// TwinCAT 3 PLC project Untitled1
// ProgramVersion: 3.1.4023.0
// libraries:
//   Tc2_MC2, * (Beckhoff Automation GmbH)
//   Tc2_Standard, * (Beckhoff Automation GmbH)
//   Tc2_System, * (Beckhoff Automation GmbH)
//   Tc3_Module, * (Beckhoff Automation GmbH)
// project tree:
//   DUTs/ stCondition.TcDUT
//   / PlcTask.TcTTO
//   POUs/ MAIN.TcPOU
// real-time tasks:
//   TASK PlcTask: cycle T#10ms, priority 20, ADS port 350
// motion (NC):
//   TASK NC-Task 1 SAF: cycle T#2ms, priority 4, ADS port 501
//   TASK NC-Task 1 SVB: cycle T#10ms, priority 8, ADS port 511
//   AXIS Axis 1 (id 1)
//     OtherSettings: AllowMotionCmdToSlave=true
//     encoder EncType=1
//     drive DrvType=5
//       Analog: TorqueSetpointScale=10, ScaleFactorActTorque=0.1
//     controller CtrType=1
//       CtrPara: PriorControlFactor=1
//         Observer: BandWidth=20
// variable links:
//   Untitled1/Untitled1 Instance <-> NC-Task 1 SAF/Axes/Axis 1
//     PlcTask Inputs/MAIN.fbAxis.NcToPlc <-> Outputs/ToPlc
//     PlcTask Outputs/MAIN.fbAxis.PlcToNc <-> Inputs/FromPlc

CONFIGURATION Untitled1
    RESOURCE PLC ON TwinCAT3
        TASK PlcTask(INTERVAL := T#10ms, PRIORITY := 20);
        PROGRAM MAIN WITH PlcTask : MAIN;
    END_RESOURCE
END_CONFIGURATION

// ---- DUTs/stCondition.TcDUT
TYPE stCondition :
STRUCT
	lrVelocity			: LREAL;
	lrAcceleration		: LREAL;
	lrDeceleration		: LREAL;
	lrJerk				: LREAL;
END_STRUCT
END_TYPE

// ---- POUs/MAIN.TcPOU
PROGRAM MAIN
VAR
	fbAxis						: AXIS_REF;
	fbPower						: MC_Power;
	fbMoveAbs_AC				: MC_MoveAbsolute;
	fbMoveAbs_CD				: MC_MoveAbsolute;
	fbMoveAbs_DE				: MC_MoveAbsolute;
	fbMoveAbs_EB				: MC_MoveAbsolute;
	fbMoveAbs_BA				: MC_MoveAbsolute;
	
	stFastCondition				: stCondition;
	stSlowCondition				: stCondition;
	
	iState						: UINT;
	bInitialized				: BOOL;
	bStartMove					: BOOL;
	
	bExeMoveAbs_AC				: BOOL;
	bExeMoveAbs_CD				: BOOL;
	bExeMoveAbs_DE				: BOOL;
	bExeMoveAbs_EB				: BOOL;
	bExeMoveAbs_BA				: BOOL;
	lrTargetPos_B				: LREAL := 500;					
END_VAR

CASE iState OF
	0: //初期化を始めますか
	IF bInitialized THEN
		iState := 10;
	END_IF
	
	10: //条件を設定します
	iState := 20;
	stFastCondition.lrVelocity := 100;
	stFastCondition.lrAcceleration := 1000;
	stFastCondition.lrDeceleration := 1000;
	stFastCondition.lrJerk := 10000;
	
	stSlowCondition.lrVelocity := 50;
	stSlowCondition.lrAcceleration := 500;
	stSlowCondition.lrDeceleration := 500;
	stSlowCondition.lrJerk := 5000;

	20: // サーボオンします
	fbPower(
		Axis:= fbAxis, 
		Enable:= TRUE, 
		Enable_Positive:= TRUE, 
		Enable_Negative:= TRUE, 
		Override:= , 
		BufferMode:= , 
		Options:= );
		
	IF fbPower.Status THEN
		//サーボオンしたら次へ
		iState := 100;
	END_IF
		
	100: //動作を開始しますか
	IF bStartMove THEN
		iState := 110;
	END_IF
	
	110: 
	IF (-0.1 < fbAxis.NcToPlc.ActPos) AND (fbAxis.NcToPlc.ActPos < 0.1) THEN
		//初期地点でAからCに移動
		bExeMoveAbs_AC := TRUE;
		bExeMoveAbs_CD := FALSE;
		bExeMoveAbs_DE := FALSE;
		bExeMoveAbs_EB := FALSE;
		bExeMoveAbs_BA := FALSE;
	ELSIF (100 < fbAxis.NcToPlc.ActPos) AND (fbAxis.NcToPlc.ActPos < 200) THEN
		// C地点についたら条件を変えてD地点に移動
		bExeMoveAbs_AC := FALSE;
		bExeMoveAbs_CD := TRUE;
		bExeMoveAbs_DE := FALSE;
		bExeMoveAbs_EB := FALSE;
		bExeMoveAbs_BA := FALSE;
	ELSIF (200 < fbAxis.NcToPlc.ActPos) AND (fbAxis.NcToPlc.ActPos < 300) THEN
		// D地点についたら条件を変えてE地点に移動
		bExeMoveAbs_AC := FALSE;
		bExeMoveAbs_CD := FALSE;
		bExeMoveAbs_DE := TRUE;
		bExeMoveAbs_EB := FALSE;
		bExeMoveAbs_BA := FALSE;
	ELSIF (300 < fbAxis.NcToPlc.ActPos) AND (fbAxis.NcToPlc.ActPos < 400) THEN
		// E地点についたら条件を変えてB地点に移動
		bExeMoveAbs_AC := FALSE;
		bExeMoveAbs_CD := FALSE;
		bExeMoveAbs_DE := FALSE;
		bExeMoveAbs_EB := TRUE;
		bExeMoveAbs_BA := FALSE;
	END_IF
	
	IF fbMoveAbs_EB.Done THEN
		//Bに到着
		iState := 120;
	END_IF

// A>C 高速条件
	fbMoveAbs_AC(
		Axis:= fbAxis, 
		Execute:= bExeMoveAbs_AC, 
		Position:= lrTargetPos_B, 
		Velocity:= stFastCondition.lrVelocity, 
		Acceleration:= stFastCondition.lrAcceleration, 
		Deceleration:= stFastCondition.lrDeceleration, 
		Jerk:= stFastCondition.lrJerk, 
		BufferMode:= , 
		Options:= );
		
	// C>D 低速条件
	fbMoveAbs_CD(
		Axis:= fbAxis, 
		Execute:= bExeMoveAbs_CD, 
		Position:= lrTargetPos_B, 
		Velocity:= stSlowCondition.lrVelocity, 
		Acceleration:= stSlowCondition.lrAcceleration, 
		Deceleration:= stSlowCondition.lrDeceleration, 
		Jerk:= stSlowCondition.lrJerk, 
		BufferMode:= , 
		Options:= );
		
	// D>E 高速条件
	fbMoveAbs_DE(
		Axis:= fbAxis, 
		Execute:= bExeMoveAbs_DE, 
		Position:= lrTargetPos_B, 
		Velocity:= stFastCondition.lrVelocity, 
		Acceleration:= stFastCondition.lrAcceleration, 
		Deceleration:= stFastCondition.lrDeceleration, 
		Jerk:= stFastCondition.lrJerk, 
		BufferMode:= , 
		Options:= );
		
	// E>B 低速条件
	fbMoveAbs_EB(
		Axis:= fbAxis, 
		Execute:= bExeMoveAbs_EB, 
		Position:= lrTargetPos_B, 
		Velocity:= stSlowCondition.lrVelocity, 
		Acceleration:= stSlowCondition.lrAcceleration, 
		Deceleration:= stSlowCondition.lrDeceleration, 
		Jerk:= stSlowCondition.lrJerk, 
		BufferMode:= , 
		Options:= );	
	
	120:
	IF fbMoveAbs_BA.Done THEN
		//Bに到着
		iState := 100;
		bExeMoveAbs_AC := FALSE;
		bExeMoveAbs_CD := FALSE;
		bExeMoveAbs_DE := FALSE;
		bExeMoveAbs_EB := FALSE;
		bExeMoveAbs_BA := FALSE;
	ELSE
		bExeMoveAbs_AC := FALSE;
		bExeMoveAbs_CD := FALSE;
		bExeMoveAbs_DE := FALSE;
		bExeMoveAbs_EB := FALSE;
		bExeMoveAbs_BA := TRUE;
	END_IF
		
	// B>A 高速条件
	fbMoveAbs_BA(
		Axis:= fbAxis, 
		Execute:= bExeMoveAbs_BA, 
		Position:= 0, 
		Velocity:= stFastCondition.lrVelocity, 
		Acceleration:= stFastCondition.lrAcceleration, 
		Deceleration:= stFastCondition.lrDeceleration, 
		Jerk:= stFastCondition.lrJerk, 
		BufferMode:= , 
		Options:= );
END_CASE

END_PROGRAM
